(* Schneider Machine Expert - Basic project PROJETO2, file version 2.9.0.0 *)
(* ProjectInformations: Name=Novo projeto *)

HARDWARE
  Cpu 0: TM200CE24R
  ModuleExtensionObject 0: TM3TI4/G
  EthernetConfiguration: NetworkName=M200, IpAllocationMode=FixedAddress, IpAddress=192.168.10.1, SubnetMask=255.255.255.0
  SerialLineConfiguration: Baud=Baud9600, Parity=ParityNone, DataBits=DataBits8, StopBits=StopBits1, PhysicalMedium=PhysicalMediumRs485, TransmissionMode=TransmissionModeModbusRtu, SlaveId=1, Addressing=SlaveAddressing
  MastTask: UsePeriodScanMode=true, PeriodScan=10
  FastTask: Period=255
  CpuBehavior: StartingMode=StartAsPreviousState, AutoSaveRamOnEeprom=true, WatchdogPeriod=250

SYMBOLS  (address, symbol, comment, settings)
  %M100     MEM_I00
  %M101     MEM_I01
  %M102     MEM_I02
  %M103     MEM_I03
  %M104     MEM_I04
  %M105     MEM_I05
  %M106     MEM_I06
  %M107     MEM_I07
  %M108     MEM_I08
  %TM0        [Preset=6]
  %TM1        [Preset=2, Base=OneSecond]
  %I0.0     DJ_GERAL_ABERTO
  %I0.1     DJ_GERAL_FECHADO
  %I0.2     RESERVA1
  %I0.3     RESERVA2
  %I0.4     RESERVA3
  %I0.5     RESERVA4
  %I0.6     RESERVA5
  %I0.7     RESERVA6
  %I0.8     RESERVA7
  %I0.9     RESERVA8
  %I0.10    STS_SERVICO_AUX
  %I0.11    BOTAO_CLOSE
  %I0.12    BOTAO_OPEN
  %I0.13    BOTAO_EMERGENCIA
  %Q0.0     COMM_OK
  %Q0.1     USINAGERANDO
  %Q0.2     FALHA
  %Q0.3     ALARME
  %Q0.4     EMERGENCIA_INV
  %Q0.5     RESET_RASP
  %Q0.6     RESET_LINK_3G
  %Q0.7     RESERVA_1
  %Q0.8     RESERVA_2
  %Q0.9     RESERVA_3
  %IW1.0    TEMP_AMBIENTE  [Type=Type_PT100, Scope=Scope_Celsius, Minimum=-2000, Maximum=8500]
  %IW1.1    TEMP_QUADRO  [Type=Type_PT100, Scope=Scope_Celsius, Minimum=-2000, Maximum=8500]
  %IW1.2    TEMP_MODULO  [Type=Type_PT100, Scope=Scope_Celsius, Minimum=-2000, Maximum=8500]
  %IW1.3    TEMP_TRAFO  [Type=Type_PT100, Scope=Scope_Celsius, Minimum=-2000, Maximum=8500]

POU Saídas
  (* SectionNumber=1 *)

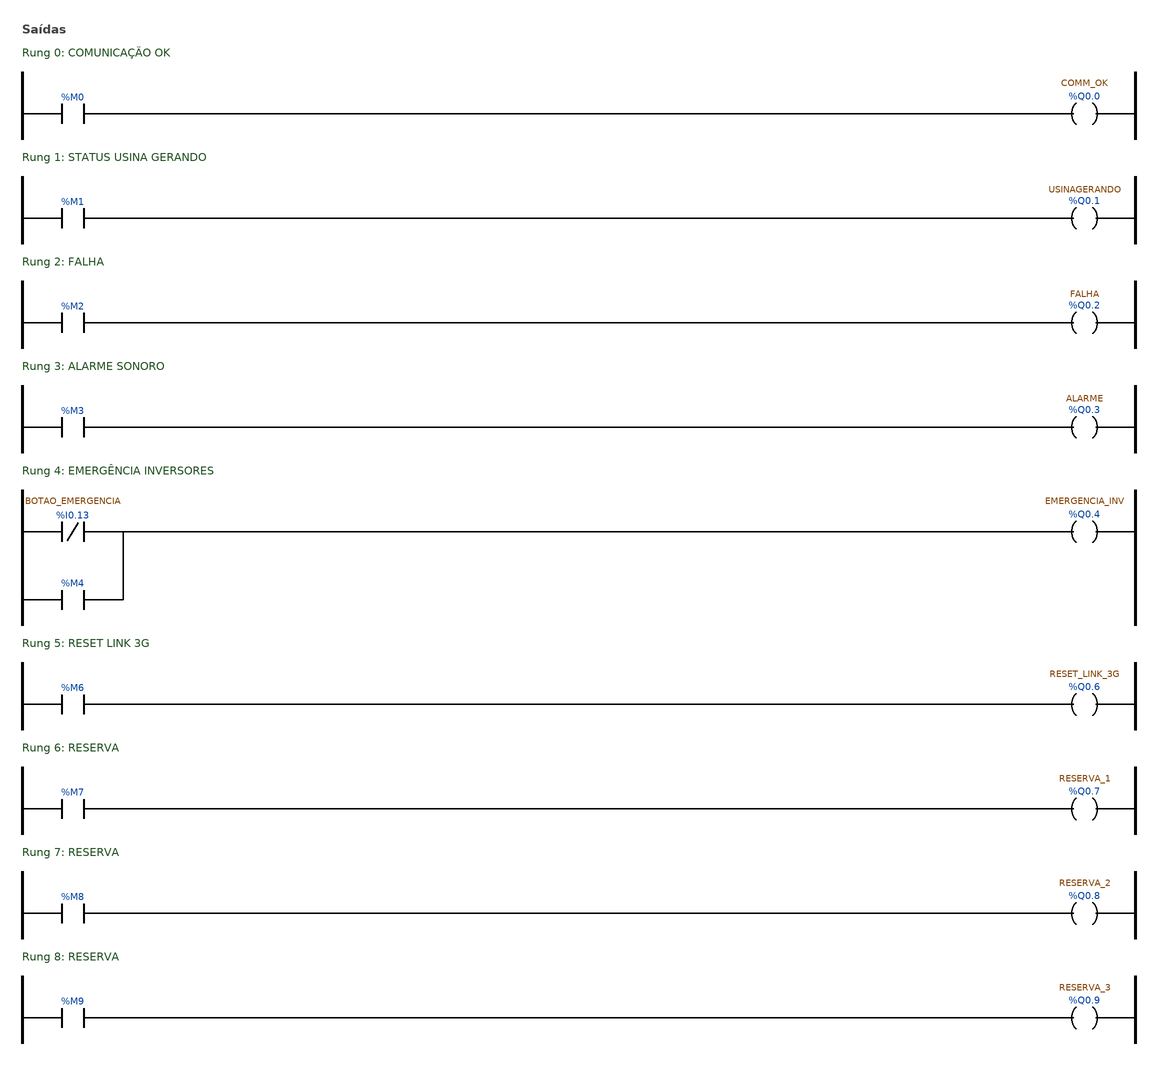

// Rung 0: COMUNICAÇÃO OK
  LD %M0
  ST %Q0.0                (* COMM_OK *)
  // as ST:
  //   COMM_OK := %M0;

// Rung 1: STATUS USINA GERANDO
  LD %M1
  ST %Q0.1                (* USINAGERANDO *)
  // as ST:
  //   USINAGERANDO := %M1;

// Rung 2: FALHA
  LD %M2
  ST %Q0.2                (* FALHA *)
  // as ST:
  //   FALHA := %M2;

// Rung 3: ALARME SONORO
  LD %M3
  ST %Q0.3                (* ALARME *)
  // as ST:
  //   ALARME := %M3;

// Rung 4: EMERGÊNCIA INVERSORES
  LDN %I0.13              (* BOTAO_EMERGENCIA *)
  OR %M4
  ST %Q0.4                (* EMERGENCIA_INV *)
  // as ST:
  //   EMERGENCIA_INV := NOT BOTAO_EMERGENCIA OR %M4;

// Rung 5: RESET LINK 3G
  LD %M6
  ST %Q0.6                (* RESET_LINK_3G *)
  // as ST:
  //   RESET_LINK_3G := %M6;

// Rung 6: RESERVA
  LD %M7
  ST %Q0.7                (* RESERVA_1 *)
  // as ST:
  //   RESERVA_1 := %M7;

// Rung 7: RESERVA
  LD %M8
  ST %Q0.8                (* RESERVA_2 *)
  // as ST:
  //   RESERVA_2 := %M8;

// Rung 8: RESERVA
  LD %M9
  ST %Q0.9                (* RESERVA_3 *)
  // as ST:
  //   RESERVA_3 := %M9;

POU Entradas
  (* SectionNumber=2 *)

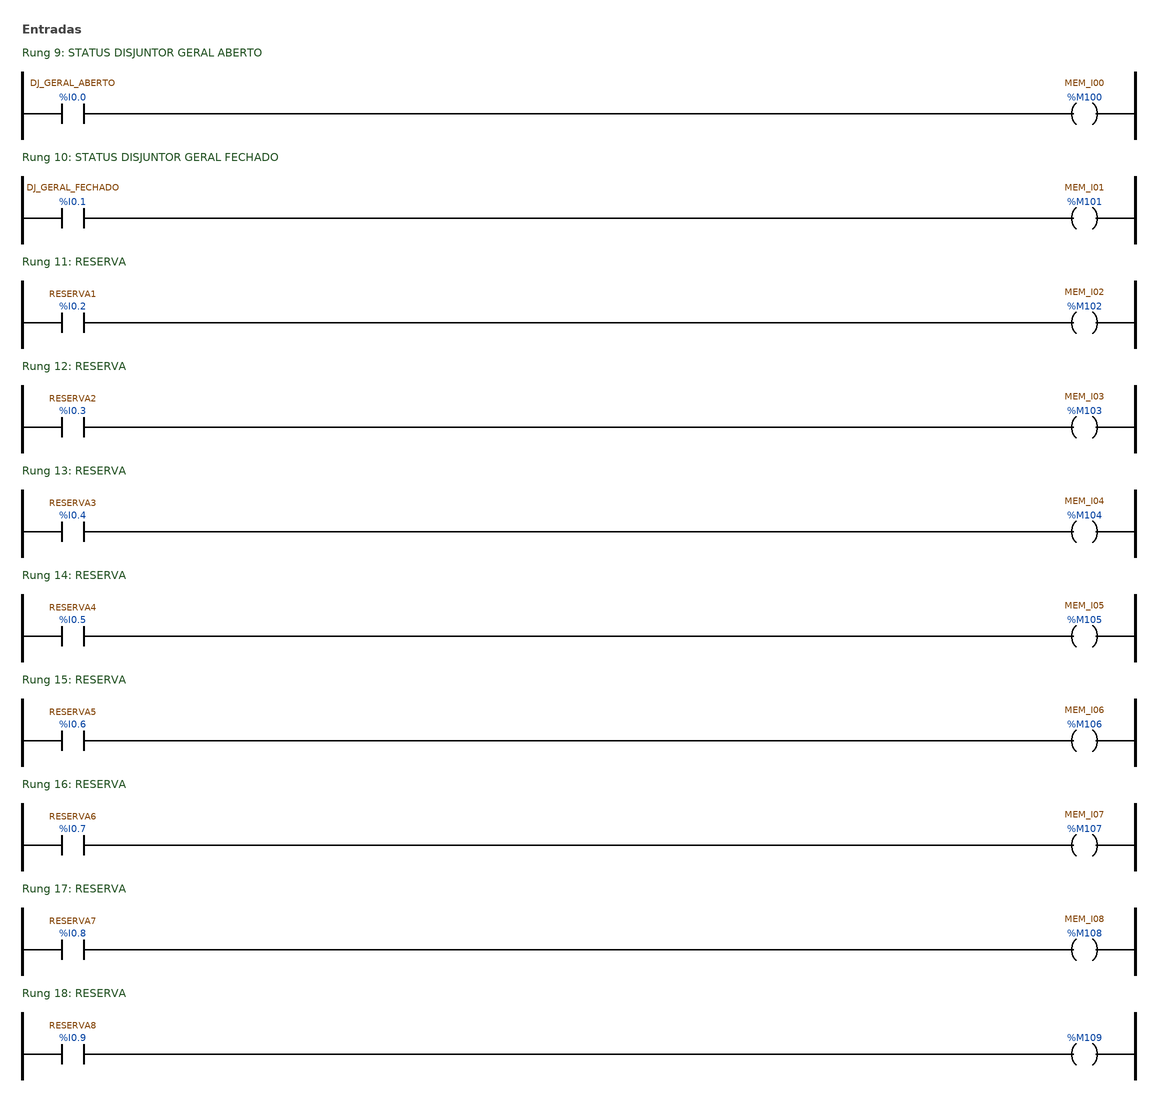

// Rung 9: STATUS DISJUNTOR GERAL ABERTO
  LD %I0.0                (* DJ_GERAL_ABERTO *)
  ST %M100                (* MEM_I00 *)
  // as ST:
  //   MEM_I00 := DJ_GERAL_ABERTO;

// Rung 10: STATUS DISJUNTOR GERAL FECHADO
  LD %I0.1                (* DJ_GERAL_FECHADO *)
  ST %M101                (* MEM_I01 *)
  // as ST:
  //   MEM_I01 := DJ_GERAL_FECHADO;

// Rung 11: RESERVA
  LD %I0.2                (* RESERVA1 *)
  ST %M102                (* MEM_I02 *)
  // as ST:
  //   MEM_I02 := RESERVA1;

// Rung 12: RESERVA
  LD %I0.3                (* RESERVA2 *)
  ST %M103                (* MEM_I03 *)
  // as ST:
  //   MEM_I03 := RESERVA2;

// Rung 13: RESERVA
  LD %I0.4                (* RESERVA3 *)
  ST %M104                (* MEM_I04 *)
  // as ST:
  //   MEM_I04 := RESERVA3;

// Rung 14: RESERVA
  LD %I0.5                (* RESERVA4 *)
  ST %M105                (* MEM_I05 *)
  // as ST:
  //   MEM_I05 := RESERVA4;

// Rung 15: RESERVA
  LD %I0.6                (* RESERVA5 *)
  ST %M106                (* MEM_I06 *)
  // as ST:
  //   MEM_I06 := RESERVA5;

// Rung 16: RESERVA
  LD %I0.7                (* RESERVA6 *)
  ST %M107                (* MEM_I07 *)
  // as ST:
  //   MEM_I07 := RESERVA6;

// Rung 17: RESERVA
  LD %I0.8                (* RESERVA7 *)
  ST %M108                (* MEM_I08 *)
  // as ST:
  //   MEM_I08 := RESERVA7;

// Rung 18: RESERVA
  LD %I0.9                (* RESERVA8 *)
  ST %M109
  // as ST:
  //   %M109 := RESERVA8;

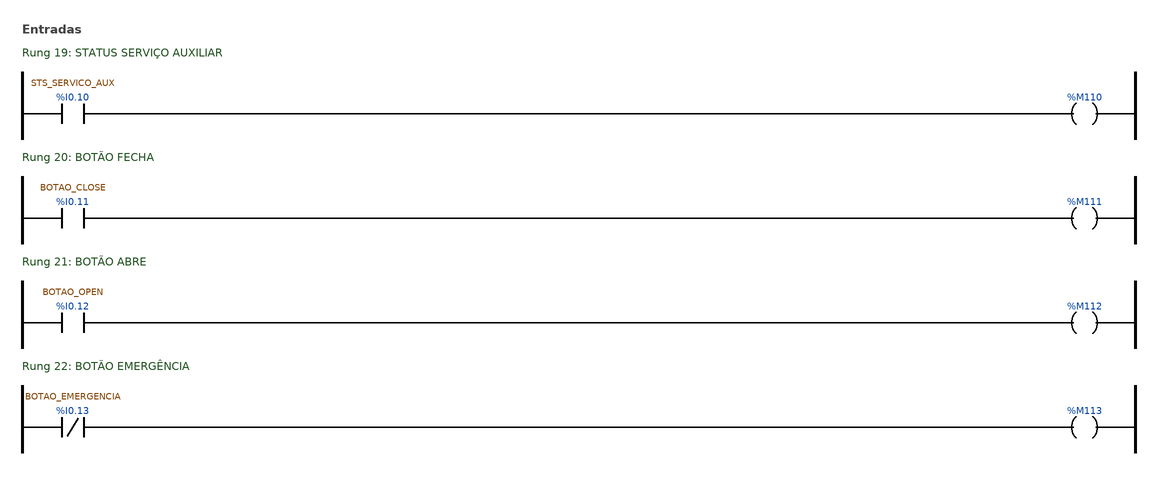

// Rung 19: STATUS SERVIÇO AUXILIAR
  LD %I0.10               (* STS_SERVICO_AUX *)
  ST %M110
  // as ST:
  //   %M110 := STS_SERVICO_AUX;

// Rung 20: BOTÃO FECHA
  LD %I0.11               (* BOTAO_CLOSE *)
  ST %M111
  // as ST:
  //   %M111 := BOTAO_CLOSE;

// Rung 21: BOTÃO ABRE
  LD %I0.12               (* BOTAO_OPEN *)
  ST %M112
  // as ST:
  //   %M112 := BOTAO_OPEN;

// Rung 22: BOTÃO EMERGÊNCIA
  LDN %I0.13              (* BOTAO_EMERGENCIA *)
  ST %M113
  // as ST:
  //   %M113 := NOT BOTAO_EMERGENCIA;

POU Analógicas
  (* SectionNumber=3 *)

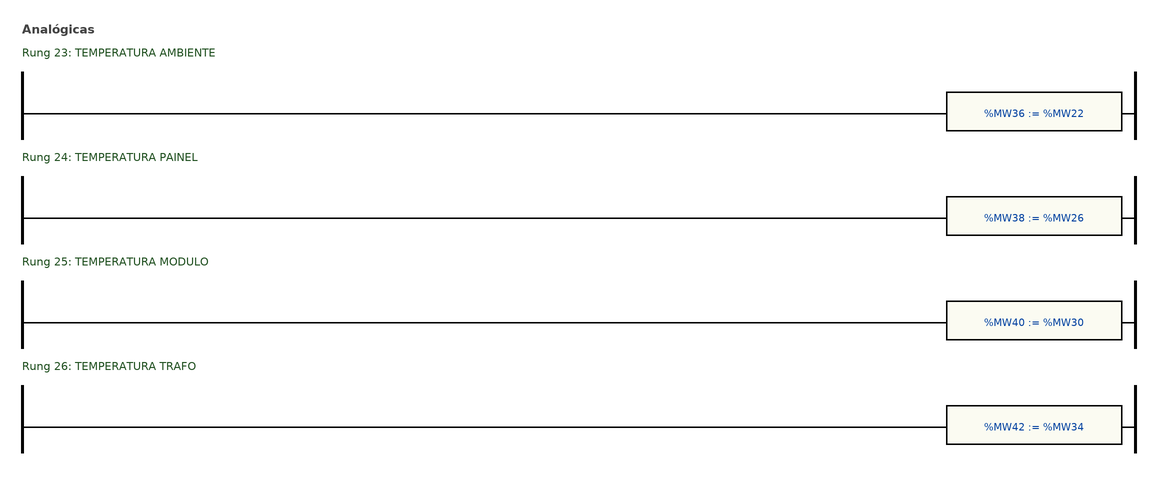

// Rung 23: TEMPERATURA AMBIENTE
  LD 1
  [ %MW36 := %MW22 ]
  // as ST:
  //   %MW36 := %MW22;

// Rung 24: TEMPERATURA PAINEL
  LD 1
  [ %MW38 := %MW26 ]
  // as ST:
  //   %MW38 := %MW26;

// Rung 25: TEMPERATURA MODULO
  LD 1
  [ %MW40 := %MW30 ]
  // as ST:
  //   %MW40 := %MW30;

// Rung 26: TEMPERATURA TRAFO
  LD 1
  [ %MW42 := %MW34 ]
  // as ST:
  //   %MW42 := %MW34;

POU ESCALA TEMPERATURA
  (* SectionNumber=4 *)

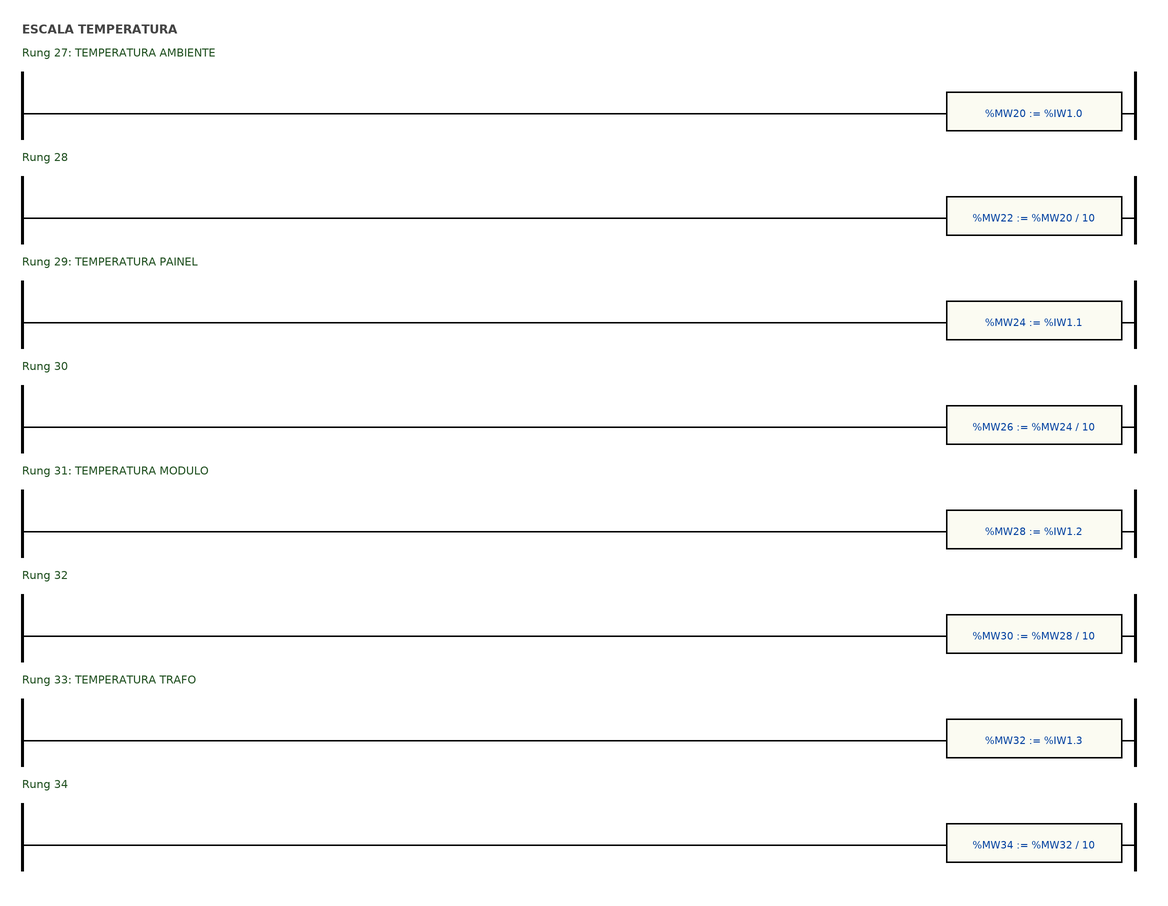

// Rung 27: TEMPERATURA AMBIENTE
  LD 1
  [ %MW20 := %IW1.0 ]     (* TEMP_AMBIENTE *)
  // as ST:
  //   %MW20 := TEMP_AMBIENTE;

// Rung 28
  LD 1
  [ %MW22 := %MW20 / 10 ]
  // as ST:
  //   %MW22 := %MW20 / 10;

// Rung 29: TEMPERATURA PAINEL
  LD 1
  [ %MW24 := %IW1.1 ]     (* TEMP_QUADRO *)
  // as ST:
  //   %MW24 := TEMP_QUADRO;

// Rung 30
  LD 1
  [ %MW26 := %MW24 / 10 ]
  // as ST:
  //   %MW26 := %MW24 / 10;

// Rung 31: TEMPERATURA MODULO
  LD 1
  [ %MW28 := %IW1.2 ]     (* TEMP_MODULO *)
  // as ST:
  //   %MW28 := TEMP_MODULO;

// Rung 32
  LD 1
  [ %MW30 := %MW28 / 10 ]
  // as ST:
  //   %MW30 := %MW28 / 10;

// Rung 33: TEMPERATURA TRAFO
  LD 1
  [ %MW32 := %IW1.3 ]     (* TEMP_TRAFO *)
  // as ST:
  //   %MW32 := TEMP_TRAFO;

// Rung 34
  LD 1
  [ %MW34 := %MW32 / 10 ]
  // as ST:
  //   %MW34 := %MW32 / 10;

POU Reset Raspberry
  (* SectionNumber=5 *)

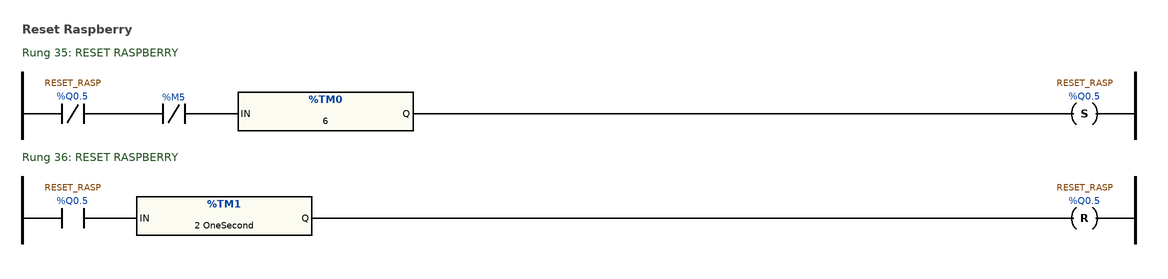

// Rung 35: RESET RASPBERRY
  BLK %TM0
  LDN %Q0.5               (* RESET_RASP *)
  ANDN %M5
  IN
  OUT_BLK
  LD Q
  S %Q0.5                 (* RESET_RASP *)
  END_BLK
  // as ST:
  //   %TM0(IN := NOT RESET_RASP AND NOT %M5);
  //   IF %TM0.Q THEN RESET_RASP := TRUE; END_IF;

// Rung 36: RESET RASPBERRY
  BLK %TM1
  LD %Q0.5                (* RESET_RASP *)
  IN
  OUT_BLK
  LD Q
  R %Q0.5                 (* RESET_RASP *)
  END_BLK
  // as ST:
  //   %TM1(IN := RESET_RASP);
  //   IF %TM1.Q THEN RESET_RASP := FALSE; END_IF;
